# EPICS IOC start-up script: ipApp/iocsh/loadSerialPort.iocsh
#- ###################################################
#- PREFIX    - IOC prefix
#- PORT      - IPAC Dev Port
#- DEVICE    - Hardware Dev Port, ex: /dev/tty0 (Default: $(PORT))
#- IN_BUFF   - Input buffer size (Default: 1000),
#- OUT_BUFF  - Output buffer size (Default:1000)
#- INSTANCE  - Instance name for asyn record (Default: asyn_$(PORT))
#- ###################################################

drvAsynSerialPortConfigure("$(PORT)", "$(DEVICE=$(PORT))", 0, 0, 0)
asynOctetConnect("$(PORT)", "$(PORT)")
dbLoadRecords("$(ASYN)/db/asynRecord.db", "P=$(PREFIX), R=$(INSTANCE=asyn_$(PORT)), PORT=$(PORT), ADDR=0, OMAX=$(OUT_BUFF=1000), IMAX=$(IN_BUFF=1000)")
